Universal Robots PolyScope program: get_data.urp

Program get_data (installation=default directory=/programs/usbdisk createdIn=3.15.4.106291 lastSavedIn=3.15.4.106291 robotSerialNumber=2019300133)
Calibrated DH parameters: a=[-0.000006, -0.606471, -0.570201, -0.000053, 0.000006, 0]; d=[0.128096, 15.114888, -22.674746, 7.723348, 0.115665, 0.092162]; alpha=[1.570605, -0.005579, -0.004649, 1.571049, -1.571015, 0]; deltaTheta=[-0.00004, -0.169247, 0.199673, -0.061563, -0.000077, -0.000043]
Robot Program (runOnlyOnce=false)
  data := [0.0, 0.0, 0.0]
  Script: camera = rpc_factory("xmlrpc","http://127.0.0.1:5000")
  Script: data = camera.get_next_pick()
  Popup Message (haltProgram=false inputType=Variable) variable=data
